PROGRAM P_VacummBeltTable
VAR
		(*Initialization*)
	bVBT_OK		: BOOL;
	bError		: BOOL;
	bStart		: BOOL;
	bStop		: BOOL;
	(*Process*)
	bVacEnable 	: BOOL;
	bVacOn		: BOOL;
	bVacOff		: BOOL;
	bOverride	: BOOL;
	(*VBT-Only Process*)
	bCuringDone	: BOOL;
	bGateCloseStatus	: BOOL;
	bBadSheetSignal		: BOOL;
	//-----------------------------------------(*Case*)-----------------------------------------------------
	
	(* Reference for VBT

	State_Init 					,
	State_AutoStart         	,
	State_AutoStop          	,
	State_AutoVacOn				,
	State_VacOff				,
	State_AutoBackToInit        ,
	State_Override				,
	State_Error		

	*)	
	
END_VAR
VAR_INPUT
	bStartCommand : BOOL;
END_VAR
VAR_OUTPUT
	iVBTcase : INT;
END_VAR

CASE iVBTcase OF
	
VacuumBeltTableState.State_Init :
	IF bVBT_OK AND bStartCommand AND 
	   (NOT bError) THEN
		iVBTcase:=VacuumBeltTableState.State_AutoStart;
	ELSE
		iVBTcase := VacuumBeltTableState.State_Init;
	END_IF
	bStart:=bStart;
	
VacuumBeltTableState.State_AutoStart :
	bStart:=TRUE;
	iVBTcase:=VacuumBeltTableState.State_AutoVacOn;
	
VacuumBeltTableState.State_AutoVacOn :
	(*Main Business logic*)
	IF NOT bError AND bCuringDone AND bGateCloseStatus THEN	
			IF bStop THEN
				iVBTcase := VacuumBeltTableState.State_VacOff;
			END_IF
		iVBTcase := iVBTcase;		
	END_IF
	IF bError THEN
		iVBTcase:=VacuumBeltTableState.State_Error;
	END_IF

	
VacuumBeltTableState.State_VacOff :
	iVBTcase:= VacuumBeltTableState.State_AutoStop;
	
VacuumBeltTableState.State_AutoStop :
	iVBTcase:= VacuumBeltTableState.State_AutoBackToInit;
	
VacuumBeltTableState.State_AutoBackToInit :
	iVBTcase := VacuumBeltTableState.State_Init;
	
VacuumBeltTableState.State_Error :
	iVBTcase:=VacuumBeltTableState.State_Init;
VacuumBeltTableState.State_Override :
	;
	//iVBTcase:=;
	
END_CASE

END_PROGRAM

(* stored: Version 1.1.0.1, ProductVersion 3.1.4024.12
   POU P_VacummBeltTable: Id {712b94c2-ba3b-4131-911d-4dda9faec154}, SpecialFunc None *)
